{attribute 'qualified_only'}
{attribute 'strict'}
TYPE E_SDSTransferArmRStates :
(
    UNKNOWN := 0,
    FULLY_CCW := 1,
    PREROTATE_SAMPLE_REMOVAL := 2,
    UNSCREW_FROM_GARAGE := 3,
    PREROTATE_SAMPLE_INSERTION := 4,
    SCREW_INTO_GARAGE := 5
) UINT;
END_TYPE

(* stored: Version 1.1.0.1
   DUT E_SDSTransferArmRStates: Id {b86e308f-2f27-08e0-1203-33ec08c41ff1} *)
